// Mitsubishi GX Works2 project: 0312_test1   PLC: Q03UDV

PROGRAM MAIN
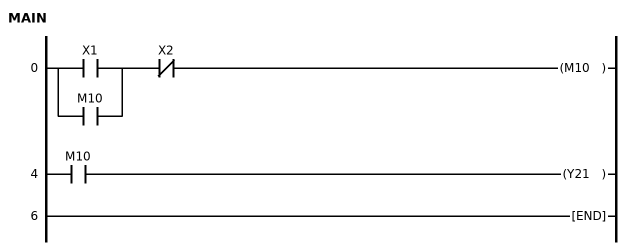
0     LD      X1
      OR      M10
      ANI     X2
      OUT     M10
4     LD      M10
      OUT     Y21
6     END
END_PROGRAM
